FUNCTION SquareSignal : REAL
VAR_INPUT
	yMin : REAL;
	yMAX : REAL;
	w : REAL;
	yOffset : REAL;
	t : REAL;
END_VAR
VAR
	reffSignal : REAL;
END_VAR

reffSignal := SIN(w*t) ;

IF(reffSignal > 0.0 ) THEN
	SquareSignal := yMAX + yOffset;
ELSIF reffSignal < 0.0 THEN
	SquareSignal := yMin + yOffset;
ELSE
	SquareSignal := 0.0;
END_IF

END_FUNCTION

(* stored: Version 1.1.0.1, ProductVersion 3.1.4022.10
   POU SquareSignal: Id {29d86ddd-4213-4211-9ca0-aef311870f69}, SpecialFunc None *)
